// TIA Portal project "washing_machine" (V18)

(* hardware
DEVICE "S7-1200 station_1"  S7-1200 Station
   slot 0: "Rack_0"  S7-1200 Rack  Rack  V1.0
   slot 1: "PLC_1"  CPU 1215C DC/DC/DC  6ES7 215-1AG40-0XB0  V4.6
*)

// ===== PLC "PLC_1"  CPU 1215C DC/DC/DC =====

VAR_GLOBAL   // PLC tag table "Default tag table"
   "start" AT %I0.0 : Bool;
   "sandık_aşağıda" AT %I0.1 : Bool;
   "sandık_yukarıda" AT %I0.2 : Bool;
   "sandık_aşağı" AT %Q0.0 : Bool;
   "sandık_yukarı" AT %Q0.1 : Bool;
   "lamba" AT %Q0.2 : Bool;
   "Tag_1" AT %M0.0 : Bool;
END_VAR

// folder: System blocks/Program resources

DATA_BLOCK "bekleme_zamanı"   // DB1
{ S7_Optimized_Access := 'TRUE' }
AUTHOR : Simatic
FAMILY : IEC
NAME : IEC_TMR
VERSION : 1.0
// stored: InstanceOfName IEC_TIMER
"IEC_TIMER"
BEGIN
END_DATA_BLOCK

DATA_BLOCK "yıkama_sayısı"   // DB2
{ S7_Optimized_Access := 'TRUE' }
AUTHOR : Simatic
FAMILY : IEC
NAME : CNTR
VERSION : 1.0
// stored: InstanceOfName IEC_COUNTER
"IEC_COUNTER"
BEGIN
END_DATA_BLOCK

// folder: (top level)

FUNCTION "Block_1" : Void   // FC1, LAD
{ S7_Optimized_Access := 'TRUE' }
VERSION : 0.1
   VAR_TEMP   // added for the SCL form of the ladder/FBD networks
      _w1 : Bool;
   END_VAR
BEGIN

REGION Network 1
   // lamba
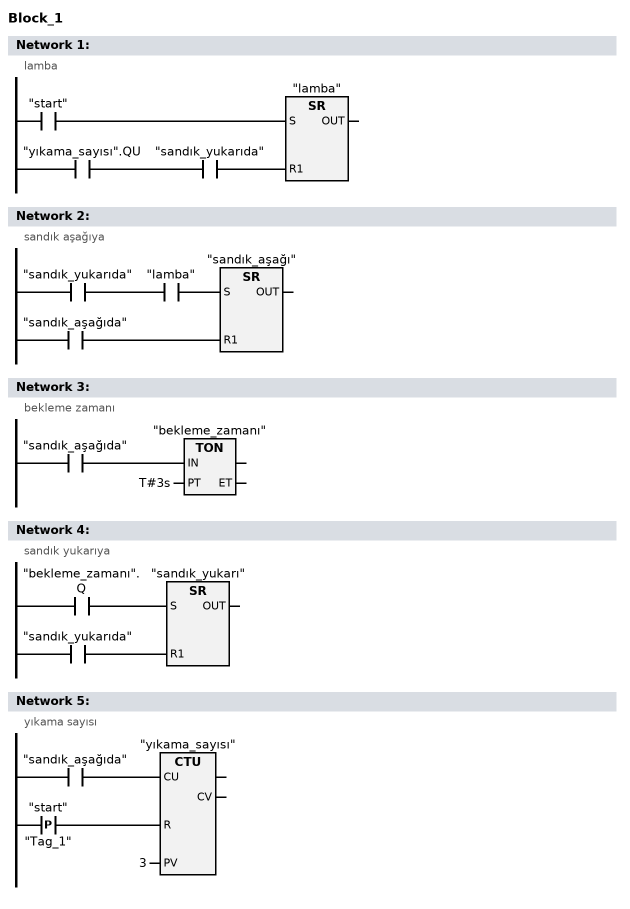
   RUNG wire#powerrail
      Contact( "start" )
      S_SR(operand := "lamba", r1 := wire#w1)
   END_RUNG
   RUNG wire#powerrail
      Contact( "yıkama_sayısı".QU )
      Contact( "sandık_yukarıda" )
   END_RUNG wire#w1
   // the same network as SCL:
   IF "start" THEN
       "lamba" := TRUE;   // SR flip-flop
   END_IF;
   IF "yıkama_sayısı".QU AND "sandık_yukarıda" THEN "lamba" := FALSE; END_IF;
END_REGION

REGION Network 2
   // sandık aşağıya
   RUNG wire#powerrail
      Contact( "sandık_yukarıda" )
      Contact( "lamba" )
      S_SR(operand := "sandık_aşağı", r1 := wire#w1)
   END_RUNG
   RUNG wire#powerrail
      Contact( "sandık_aşağıda" )
   END_RUNG wire#w1
   // the same network as SCL:
   IF "sandık_yukarıda" AND "lamba" THEN
       "sandık_aşağı" := TRUE;   // SR flip-flop
   END_IF;
   IF "sandık_aşağıda" THEN "sandık_aşağı" := FALSE; END_IF;
END_REGION

REGION Network 3
   // bekleme zamanı
   "bekleme_zamanı".TON(IN := "sandık_aşağıda", PT := T#3s);
END_REGION

REGION Network 4
   // sandık yukarıya
   RUNG wire#powerrail
      Contact( "bekleme_zamanı".Q )
      S_SR(operand := "sandık_yukarı", r1 := wire#w1)
   END_RUNG
   RUNG wire#powerrail
      Contact( "sandık_yukarıda" )
   END_RUNG wire#w1
   // the same network as SCL:
   IF "bekleme_zamanı".Q THEN
       "sandık_yukarı" := TRUE;   // SR flip-flop
   END_IF;
   IF "sandık_yukarıda" THEN "sandık_yukarı" := FALSE; END_IF;
END_REGION

REGION Network 5
   // yıkama sayısı
   #_w1 := "start" AND NOT "Tag_1";   // rising edge of "start"
   "Tag_1" := "start";
   "yıkama_sayısı".CTU(CU := "sandık_aşağıda", R := #_w1, PV := 3);
END_REGION
END_FUNCTION

ORGANIZATION_BLOCK "Main"   // OB1, LAD, ProgramCycle
TITLE = "Main Program Sweep (Cycle)"
{ S7_Optimized_Access := 'TRUE' }
VERSION : 0.1
   VAR_INPUT
      Initial_Call : Bool;   // Initial call of this OB
      Remanence : Bool;   // =True, if remanent data are available
   END_VAR
BEGIN

REGION Network 1
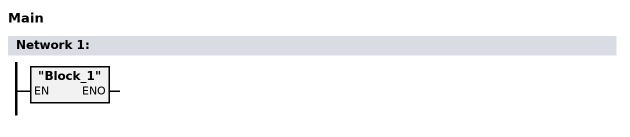
   RUNG wire#powerrail
      "Block_1"()
   END_RUNG
   // the same network as SCL:
   "Block_1"();
END_REGION
END_ORGANIZATION_BLOCK